// TIA Portal project "Logic Gates" (V16)

(* hardware
DEVICE "S7300/ET200M station_1"  S7-300 station
   slot 0: "Rail_0"  Rail  6ES7 390-1***0-0AA0
   slot 2: "PLC_1"  CPU 313C-2 DP  6ES7 313-6CF03-0AB0  V2.6
      slot 0: "MPI interface_1"  X1
      slot 1: "DP interface_1"  X2
      slot 2: "DI 16/DO 16_1"  DI16/DO16
      slot 4: "Count_1"  Counter
*)

// ===== PLC "PLC_1"  CPU 313C-2 DP =====

VAR_GLOBAL   // PLC tag table "Default tag table_1"
   "A" AT %I0.0 : Bool;
   "B" AT %I0.1 : Bool;
   "O/P" AT %Q0.0 : Bool;
   "C" AT %I0.2 : Bool;
   "D" AT %I0.3 : Bool;
END_VAR

ORGANIZATION_BLOCK "Main"   // OB1, LAD
TITLE = "Main Program Sweep (Cycle)"
{ S7_Optimized_Access := 'FALSE' }
VERSION : 0.1
   VAR_TEMP
      OB1_EV_CLASS : Byte;   // Bits 0-3 = 1 (Coming event), Bits 4-7 = 1 (Event class 1)
      OB1_SCAN_1 : Byte;   // 1 (Cold restart scan 1 of OB 1), 3 (Scan 2-n of OB 1)
      OB1_PRIORITY : Byte;   // Priority of OB Execution
      OB1_OB_NUMBR : Byte;   // 1 (Organization block 1, OB1)
      OB1_RESERVED_1 : Byte;   // Reserved for system
      OB1_RESERVED_2 : Byte;   // Reserved for system
      OB1_PREV_CYCLE : Int;   // Cycle time of previous OB1 scan (milliseconds)
      OB1_MIN_CYCLE : Int;   // Minimum cycle time of OB1 (milliseconds)
      OB1_MAX_CYCLE : Int;   // Maximum cycle time of OB1 (milliseconds)
      OB1_DATE_TIME : Date_And_Time;   // Date and time OB1 started
   END_VAR
BEGIN

REGION Network 1: AND Gate
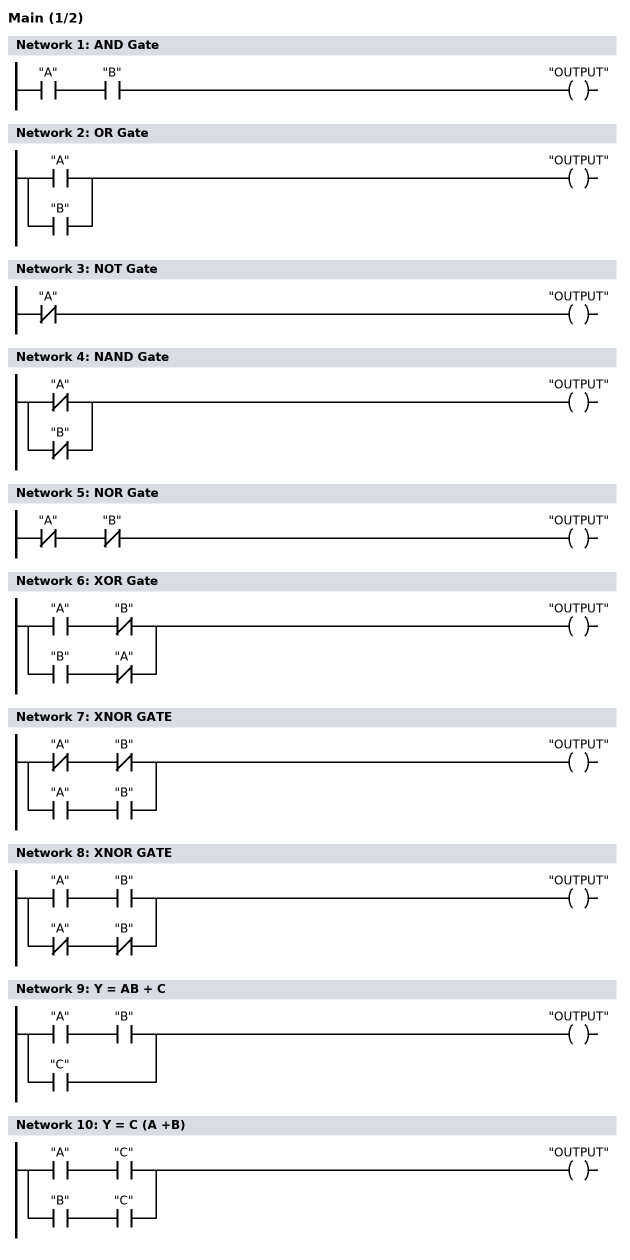
   RUNG wire#powerrail
      Contact( "A" )
      Contact( "B" )
      Coil( "OUTPUT" )
   END_RUNG
   // the same network as SCL:
   "OUTPUT" := "A" AND "B";
END_REGION

REGION Network 2: OR Gate
   RUNG wire#powerrail
      Contact( "A" )
      wire#w1
      Coil( "OUTPUT" )
   END_RUNG
   RUNG wire#powerrail
      Contact( "B" )
   END_RUNG wire#w1
   // the same network as SCL:
   "OUTPUT" := "A" OR "B";
END_REGION

REGION Network 3: NOT Gate
   RUNG wire#powerrail
      I_Contact( "A" )
      Coil( "OUTPUT" )
   END_RUNG
   // the same network as SCL:
   "OUTPUT" := NOT "A";
END_REGION

REGION Network 4: NAND Gate
   RUNG wire#powerrail
      I_Contact( "A" )
      wire#w1
      Coil( "OUTPUT" )
   END_RUNG
   RUNG wire#powerrail
      I_Contact( "B" )
   END_RUNG wire#w1
   // the same network as SCL:
   "OUTPUT" := NOT "A" OR NOT "B";
END_REGION

REGION Network 5: NOR Gate
   RUNG wire#powerrail
      I_Contact( "A" )
      I_Contact( "B" )
      Coil( "OUTPUT" )
   END_RUNG
   // the same network as SCL:
   "OUTPUT" := NOT "A" AND NOT "B";
END_REGION

REGION Network 6: XOR Gate
   RUNG wire#powerrail
      Contact( "A" )
      I_Contact( "B" )
      wire#w1
      Coil( "OUTPUT" )
   END_RUNG
   RUNG wire#powerrail
      Contact( "B" )
      I_Contact( "A" )
   END_RUNG wire#w1
   // the same network as SCL:
   "OUTPUT" := ("A" AND NOT "B") OR ("B" AND NOT "A");
END_REGION

REGION Network 7: XNOR GATE
   RUNG wire#powerrail
      I_Contact( "A" )
      I_Contact( "B" )
      wire#w1
      Coil( "OUTPUT" )
   END_RUNG
   RUNG wire#powerrail
      Contact( "A" )
      Contact( "B" )
   END_RUNG wire#w1
   // the same network as SCL:
   "OUTPUT" := (NOT "A" AND NOT "B") OR ("A" AND "B");
END_REGION

REGION Network 8: XNOR GATE
   RUNG wire#powerrail
      Contact( "A" )
      Contact( "B" )
      wire#w1
      Coil( "OUTPUT" )
   END_RUNG
   RUNG wire#powerrail
      I_Contact( "A" )
      I_Contact( "B" )
   END_RUNG wire#w1
   // the same network as SCL:
   "OUTPUT" := ("A" AND "B") OR (NOT "A" AND NOT "B");
END_REGION

REGION Network 9: Y = AB + C
   RUNG wire#powerrail
      Contact( "A" )
      Contact( "B" )
      wire#w1
      Coil( "OUTPUT" )
   END_RUNG
   RUNG wire#powerrail
      Contact( "C" )
   END_RUNG wire#w1
   // the same network as SCL:
   "OUTPUT" := ("A" AND "B") OR "C";
END_REGION

REGION Network 10: Y = C (A +B)
   RUNG wire#powerrail
      Contact( "A" )
      Contact( "C" )
      wire#w1
      Coil( "OUTPUT" )
   END_RUNG
   RUNG wire#powerrail
      Contact( "B" )
      Contact( "C" )
   END_RUNG wire#w1
   // the same network as SCL:
   "OUTPUT" := ("A" AND "C") OR ("B" AND "C");
END_REGION

REGION Network 11: Y = (AB +CD)
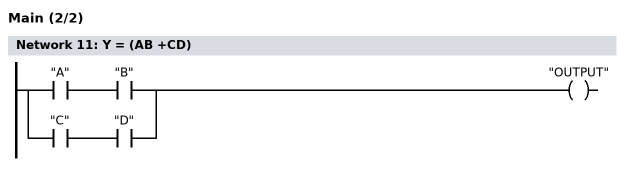
   RUNG wire#powerrail
      Contact( "A" )
      Contact( "B" )
      wire#w1
      Coil( "OUTPUT" )
   END_RUNG
   RUNG wire#powerrail
      Contact( "C" )
      Contact( "D" )
   END_RUNG wire#w1
   // the same network as SCL:
   "OUTPUT" := ("A" AND "B") OR ("C" AND "D");
END_REGION
END_ORGANIZATION_BLOCK